(* IEC 61131-3 sources: Word/plc-course/04-ladder-logic/labs/solutions, 4 files *)

(* ---- 04-1-start-stop-station.st ---- *)
(* Lab 04-1: Start/stop from two stations (local and remote).
   Module 04 (Ladder logic fundamentals).
   REFERENCE SOLUTION - try the lab yourself first.
   The same logic drawn as ladder rungs is in the Module 04 README (Lab 04-1).
   Training exercise only: emergency stops are hard-wired or use
   safety-rated devices (Module 20). *)

PROGRAM TwoStationStart
  VAR (* I/O - addresses follow the OpenPLC convention *)
    LocalStartPB    AT %IX0.0 : BOOL;  (* Start at the local station beside the pump, NO: TRUE while pressed *)
    LocalStopPB_NC  AT %IX0.1 : BOOL;  (* Stop at the local station, NC: TRUE while NOT pressed *)
    RemoteStartPB   AT %IX0.2 : BOOL;  (* Start on the control-room panel, NO: TRUE while pressed *)
    RemoteStopPB_NC AT %IX0.3 : BOOL;  (* Stop on the control-room panel, NC: TRUE while NOT pressed *)
    Motor           AT %QX0.0 : BOOL;  (* Pump motor contactor coil *)
    RunLamp         AT %QX0.1 : BOOL;  (* "Running" lamp *)
    StoppedLamp     AT %QX0.2 : BOOL;  (* "Stopped" lamp *)
  END_VAR

  (* Rung 1 - pump motor, seal-in from two stations.
     Starts in PARALLEL (OR): either station can start the pump, and the
     motor's own bit in parallel with them holds it on (the seal-in).
     Stops in SERIES (AND): either station can stop it.
     Both stop buttons are wired NC, so each reads TRUE while it is healthy
     and not pressed. They are examined with NORMALLY-OPEN contacts in ladder
     (XIC), which is why there is no NOT in front of them here.
     The stops are outside the OR, so a stop beats a start that is held at
     the other station (stop-dominant). *)
  Motor := (LocalStartPB OR RemoteStartPB OR Motor)
           AND LocalStopPB_NC AND RemoteStopPB_NC;

  (* Rungs 2 and 3 - lamps. They come after rung 1, so they show the motor
     state from THIS scan, not the previous one. StoppedLamp uses a
     normally-closed contact on an internal bit: here NOT is exactly right. *)
  RunLamp := Motor;
  StoppedLamp := NOT Motor;
END_PROGRAM

CONFIGURATION Config0
  RESOURCE Res0 ON PLC
    TASK MainTask(INTERVAL := T#10ms, PRIORITY := 0);
    PROGRAM Inst0 WITH MainTask : TwoStationStart;
  END_RESOURCE
END_CONFIGURATION

(* ---- 04-2-forward-reverse.st ---- *)
(* Lab 04-2: Forward/reverse motor with interlocks and travel limits.
   Module 04 (Ladder logic fundamentals).
   REFERENCE SOLUTION - try the lab yourself first.
   The same logic drawn as ladder rungs is in the Module 04 README (Lab 04-2).
   The software interlock here does NOT replace the electrical interlock
   (auxiliary NC contacts) and the mechanical interlock of the reversing
   contactor pair: a real starter has all three. Training exercise only. *)

PROGRAM ForwardReverse
  VAR (* I/O - addresses follow the OpenPLC convention *)
    FwdPB         AT %IX0.0 : BOOL;  (* Forward push-button, NO: TRUE while pressed *)
    RevPB         AT %IX0.1 : BOOL;  (* Reverse push-button, NO: TRUE while pressed *)
    StopPB_NC     AT %IX0.2 : BOOL;  (* Stop push-button, NC: TRUE while NOT pressed *)
    FwdLimitOK_NC AT %IX0.3 : BOOL;  (* Forward end-of-travel limit switch, NC: TRUE while NOT at the limit *)
    RevLimitOK_NC AT %IX0.4 : BOOL;  (* Reverse end-of-travel limit switch, NC: TRUE while NOT at the limit *)
    OverloadOK_NC AT %IX0.5 : BOOL;  (* Overload relay auxiliary contact, NC: TRUE while healthy *)
    FwdK          AT %QX0.0 : BOOL;  (* Forward contactor coil *)
    RevK          AT %QX0.1 : BOOL;  (* Reverse contactor coil *)
  END_VAR

  (* Rung 1 - FORWARD contactor.
     Start branch: FwdPB AND NOT RevPB. If both direction buttons are pressed
     together the command is ambiguous, so neither direction starts. Without
     this, rung order would decide: forward would always win.
     Seal-in: FwdK in parallel with the start branch.
     In series with everything (they break the seal-in):
       - StopPB_NC and OverloadOK_NC stop both directions;
       - FwdLimitOK_NC stops FORWARD only, so the operator can still reverse
         away from the forward limit;
       - NOT RevK is the software interlock: forward cannot start while
         reverse is on. The operator must stop before changing direction. *)
  FwdK := ((FwdPB AND NOT RevPB) OR FwdK)
          AND StopPB_NC AND OverloadOK_NC AND FwdLimitOK_NC AND NOT RevK;

  (* Rung 2 - REVERSE contactor, the mirror image of rung 1.
     NOT FwdK reads the value rung 1 has just written in this scan, so the
     two contactors can never both be TRUE at the end of a scan. *)
  RevK := ((RevPB AND NOT FwdPB) OR RevK)
          AND StopPB_NC AND OverloadOK_NC AND RevLimitOK_NC AND NOT FwdK;
END_PROGRAM

CONFIGURATION Config0
  RESOURCE Res0 ON PLC
    TASK MainTask(INTERVAL := T#10ms, PRIORITY := 0);
    PROGRAM Inst0 WITH MainTask : ForwardReverse;
  END_RESOURCE
END_CONFIGURATION

(* ---- 04-3-jog-run.st ---- *)
(* Lab 04-3: Jog/run selector.
   Module 04 (Ladder logic fundamentals).
   REFERENCE SOLUTION - try the lab yourself first.
   The same logic drawn as ladder rungs is in the Module 04 README (Lab 04-3).
   Training exercise only: on a real machine, jogging with guards open is a
   safety function with its own rules (reduced speed, hold-to-run devices,
   enabling devices) and safety-rated hardware (Modules 19 and 20). *)

PROGRAM JogRun
  VAR (* I/O - addresses follow the OpenPLC convention *)
    StartPB       AT %IX0.0 : BOOL;  (* Start push-button, NO: TRUE while pressed *)
    StopPB_NC     AT %IX0.1 : BOOL;  (* Stop push-button, NC: TRUE while NOT pressed *)
    JogPB         AT %IX0.2 : BOOL;  (* Jog push-button, NO: TRUE while pressed *)
    RunSel        AT %IX0.3 : BOOL;  (* JOG/RUN selector: TRUE = RUN, FALSE = JOG *)
    OverloadOK_NC AT %IX0.4 : BOOL;  (* Overload relay auxiliary contact, NC: TRUE while healthy *)
    Motor         AT %QX0.0 : BOOL;  (* Conveyor motor contactor coil *)
    RunLamp       AT %QX0.1 : BOOL;  (* "Running" lamp: continuous run only, not jogging *)
  END_VAR
  VAR (* internal *)
    RunLatch : BOOL;  (* continuous-run memory: the ONLY bit that seals in *)
    JogCmd   : BOOL;  (* jog command: never sealed in *)
  END_VAR

  (* Rung 1 - continuous run. A normal seal-in, but it seals on its own
     internal bit RunLatch, NOT on the Motor output. RunSel is in series with
     the whole rung, so switching to JOG drops the latch, and switching back
     to RUN needs a new Start. *)
  RunLatch := (StartPB OR RunLatch) AND RunSel AND StopPB_NC AND OverloadOK_NC;

  (* Rung 2 - jog. Only in JOG mode, only while the button is held, and the
     same stop and overload conditions apply. There is no seal-in contact on
     this rung at all: that is what makes it a jog. *)
  JogCmd := JogPB AND NOT RunSel AND StopPB_NC AND OverloadOK_NC;

  (* Rung 3 - the motor output is driven from ONE place: run OR jog.
     Nothing reads Motor back as a seal-in, so a jog can never latch. *)
  Motor := RunLatch OR JogCmd;

  (* Rung 4 - the lamp shows continuous running only. *)
  RunLamp := RunLatch;
END_PROGRAM

CONFIGURATION Config0
  RESOURCE Res0 ON PLC
    TASK MainTask(INTERVAL := T#10ms, PRIORITY := 0);
    PROGRAM Inst0 WITH MainTask : JogRun;
  END_RESOURCE
END_CONFIGURATION

(* ---- 04-4-tank-fill.st ---- *)
(* Lab 04-4: Tank fill valve with set/reset (latch/unlatch).
   Module 04 (Ladder logic fundamentals).
   REFERENCE SOLUTION - try the lab yourself first.
   The same logic drawn as ladder rungs is in the Module 04 README (Lab 04-4).
   Training exercise only: overfill protection that matters for safety or
   the environment is a separate, independent function (Module 20). *)

PROGRAM TankFill
  VAR (* I/O - addresses follow the OpenPLC convention *)
    AutoSel        AT %IX0.0 : BOOL;  (* OFF/AUTO selector: TRUE = AUTO *)
    LevelAboveLow  AT %IX0.1 : BOOL;  (* LSL-101 low level switch: TRUE while the level is ABOVE it (switch covered) *)
    HighLevelOK_NC AT %IX0.2 : BOOL;  (* LSH-102 high level switch, NC: TRUE while the level is BELOW it; FALSE at high level or broken wire *)
    ResetPB        AT %IX0.3 : BOOL;  (* Fault reset push-button, NO: TRUE while pressed *)
    FillValve      AT %QX0.0 : BOOL;  (* XV-100 inlet valve solenoid: TRUE = open (spring return, fail closed) *)
    SensorFault    AT %QX0.1 : BOOL;  (* Amber lamp: level switches disagree (latched) *)
  END_VAR
  VAR (* internal *)
    SwitchesDisagree : BOOL;  (* low switch says "low" while high switch says "high": impossible *)
    FaultLatch       : SR;    (* IEC SR = SET-dominant bistable (input S1 wins) *)
  END_VAR
  (* FillValve and FaultLatch are deliberately NOT retentive: after any
     restart the valve starts closed and waits for the low switch. *)

  (* Rung 1 - plausibility check. The level cannot be below the low switch
     and above the high switch at the same time, so one of the two switches
     (or its wiring) is wrong. *)
  SwitchesDisagree := NOT LevelAboveLow AND NOT HighLevelOK_NC;

  (* Rung 2 - fault latch, SET-dominant: while the disagreement is still
     there, holding Reset cannot clear it. *)
  FaultLatch(S1 := SwitchesDisagree, R := ResetPB);
  SensorFault := FaultLatch.Q1;

  (* Rung 3 - SET (latch) the valve: AUTO and the level has fallen below the
     low switch. Like a set coil, this only ever writes TRUE. *)
  IF AutoSel AND NOT LevelAboveLow THEN
    FillValve := TRUE;
  END_IF;

  (* Rung 4 - RESET (unlatch) the valve: high level reached, AUTO switched
     off, or a sensor fault. Like a reset coil, this only ever writes FALSE.
     It comes AFTER the set rung, so if both are true in the same scan the
     reset wins (last write wins): high level always closes the valve. *)
  IF NOT HighLevelOK_NC OR NOT AutoSel OR SensorFault THEN
    FillValve := FALSE;
  END_IF;
END_PROGRAM

CONFIGURATION Config0
  RESOURCE Res0 ON PLC
    TASK MainTask(INTERVAL := T#10ms, PRIORITY := 0);
    PROGRAM Inst0 WITH MainTask : TankFill;
  END_RESOURCE
END_CONFIGURATION
